// function to house all commmands to do with idx motor 

FUNCTION_BLOCK IDXMotor
VAR_INPUT
	//
END_VAR
VAR_OUTPUT
END_VAR
VAR
	Axis: AXIS_REF;
	Enabled: BOOL := FALSE;
	Override: LREAL:=100;
	MotorError AT%I*	:WORD;
	MotorErrorSent : WORD;
	AxisErrorSent:UDINT;
	NCError : WORD;
	fbMessage : FB_TcMessage;
	EnableEventSent:BOOL:= TRUE;
	HomeEventSent:BOOL:=TRUE;
    fbAxisMoveAbsolute: MC_MoveAbsolute;	
	fbMcHome: MC_Home;
	fbAxisPower: MC_Power;
	fbReset: MC_Reset;
	fbMoveRel : MC_MoveRelative;
	
END_VAR

Axis.ReadStatus();

// cyclic events below 

IF NOT (MotorError = MotorErrorSent) THEN// Creates Event 
	MotorErrorSent:= MotorError;
	fbMessage.CreateEx(TC_Events.LinearMotor.IDXmotorError,0);
	fbMessage.ipArguments.Clear().AddDWord(MotorError);
	fbMessage.Send(0);
END_IF

IF NOT (Axis.NcToPlc.ErrorCode = AxisErrorSent) THEN// Creates Event 
	AxisErrorSent:= Axis.NcToPlc.ErrorCode;
	fbMessage.CreateEx(TC_Events.LinearMotor.AxisError,0);
	fbMessage.ipArguments.Clear().AddDWord(Axis.NcToPlc.ErrorCode);
	fbMessage.Send(0);
END_IF

METHOD PUBLIC Enable : BOOL
VAR_INPUT
EnableMotor :BOOL;
END_VAR
	fbAxisPower( // use in idx class
    Axis:= Axis,
    Enable:= EnableMotor,
    Enable_Positive:= EnableMotor,
    Enable_Negative:= EnableMotor,
    Override:= Override,
	Status=>Enable,
	Error=>
);
	
	
IF EnableMotor = EnableEventSent THEN	
	EnableEventSent := NOT EnableEventSent;
IF EnableMotor THEN
	fbMessage.CreateEx(TC_Events.LinearMotor.Motor_enabled,0);
ELSE
	fbMessage.CreateEx(TC_Events.LinearMotor.Motor_disabled,0);
END_IF
fbMessage.Send(0);
END_IF
END_METHOD

METHOD Estop : BOOL
VAR_INPUT
END_VAR
//stop motor mc stop
END_METHOD

METHOD FB_init : BOOL
VAR_INPUT
	bInitRetains : BOOL; // if TRUE, the retain variables are initialized (warm start / cold start)
	bInCopyCode : BOOL;  // if TRUE, the instance afterwards gets moved into the copy code (online change)
	//AXIS_REF :REFERENCE TO AXIS_REF;
END_VAR
//Axis :=AXIS_REF;
fbMessage.CreateEx(TC_Events.LinearMotor.PLC_restarted,0);
	fbMessage.Send(0);
END_METHOD

METHOD PUBLIC Home : BOOL
VAR_IN_OUT
	Execute:BOOL;
END_VAR
VAR
	HomingDone:BOOL;
	HomingError:BOOL;
	HomingErrorID:UDINT;
END_VAR
// try changing limits to no error mode then home 


	fbMcHome(
	Axis:=Axis,
	Execute:=Execute,
	Position:=510,
	HomingMode:=MC_DefaultHoming,
	Busy=>Home,
	Done=>HomingDone,
	Error=> HomingError,
	ErrorID=> HomingErrorID
);
	
IF Execute THEN
	HomeEventSent:= FALSE;
	fbMessage.CreateEx(TC_Events.LinearMotor.Homing,0);
	fbMessage.Send(0);
	Execute:= FALSE;	
END_IF
IF HomingDone THEN
	fbMessage.CreateEx(TC_Events.LinearMotor.HomingComplete,0);
	fbMessage.Send(0);
END_IF

IF HomingError THEN
	fbMessage.CreateEx(TC_Events.LinearMotor.HomingFailed,0);
	fbMessage.ipArguments.Clear().AddDWord(HomingErrorID);
	fbMessage.Send(0);
END_IF
END_METHOD

METHOD PUBLIC Homed : BOOL
VAR_INPUT
END_VAR
Homed:=Axis.NcToPlc.StateDWord.1;
END_METHOD

METHOD MoveRelative : BOOL
VAR_INPUT
	Distance: LREAL;
	Velocity: LREAL;	
END_VAR
VAR_IN_OUT
	Execute: BOOL;
END_VAR
	fbMoveRel( // in idx class 
    Axis:= Axis,
    Execute:= Execute,
    Distance:= Distance,
    Velocity:= Velocity,);
	
		IF Execute THEN
	fbMessage.CreateEx(TC_Events.LinearMotor.RelativeMove,0);
	fbMessage.ipArguments.Clear();
	fbMessage.ipArguments.AddLReal(Distance);
	fbMessage.ipArguments.AddLReal(Velocity);
	fbMessage.Send(0);
	Execute := FALSE;
END_IF

IF fbMoveRel.Done  THEN
	fbMessage.CreateEx(TC_Events.LinearMotor.MoveComplete,0);
	fbMessage.Send(0);
	
END_IF
END_METHOD

METHOD MoveTo : BOOL
VAR_INPUT
	Position: LREAL;
	Velocity: LREAL;	
END_VAR
VAR_IN_OUT
		Execute: BOOL;
END_VAR
	fbAxisMoveAbsolute( // in idx class 
    Axis:= Axis,
    Execute:= Execute,
    Position:= Position,
    Velocity:= Velocity,);
	
	IF Execute THEN
	fbMessage.CreateEx(TC_Events.LinearMotor.MotorMove,0);
	fbMessage.ipArguments.Clear();
	fbMessage.ipArguments.AddLReal(Position);
	fbMessage.ipArguments.AddLReal(Velocity);
	fbMessage.Send(0);
	Execute := FALSE;

END_IF

IF fbAxisMoveAbsolute.Done  THEN
	fbMessage.CreateEx(TC_Events.LinearMotor.MoveComplete,0);
	fbMessage.Send(0);

	
END_IF
END_METHOD

METHOD Position : LReal
VAR_INPUT
END_VAR
Position:= Axis.NcToPlc.ActPos;
END_METHOD

METHOD Reset : BOOL
VAR_IN_OUT
	ResetAxis:BOOL;
	IDXControlByte1 :USINT;
END_VAR
fbReset(
Axis:=Axis,
Execute:=ResetAxis,
Done =>Reset);

IF resetAxis THEN
IDXControlByte1 := 16#80;// restop linear Motor
fbMessage.CreateEx(TC_Events.LinearMotor.AxisReset,0);
fbMessage.send(0);
resetAxis := FALSE;
END_IF
END_METHOD

METHOD SetSpeed : BOOL
VAR_INPUT
END_VAR
END_METHOD

METHOD PUBLIC Status : ST_AxisStatus
VAR_INPUT
END_VAR
Status := Axis.Status;
END_METHOD

END_FUNCTION_BLOCK

(* stored: Version 1.1.0.1, ProductVersion 3.1.4024.11
   POU IDXMotor: Id {2d0ab0a1-a5a3-4c64-bc51-ecb0c0b67505}, SpecialFunc None
   Method Enable: Id {6ca24d5a-5a8e-43ff-a8c3-908b75374a87}
   Method Estop: Id {ac352b5d-b443-47be-8d49-18781876fd67}
   Method FB_init: Id {98ef687f-1654-43bd-b72b-b96bfe4346b9}
   Method Home: Id {dadfc02e-e1cb-43e2-bcd9-54c8e8b7850a}
   Method Homed: Id {c1cc68f4-37cf-40df-838e-d05e58b07ab5}
   Method MoveRelative: Id {b8493f8e-43b3-46fb-816b-e627b7c74ccc}
   Method MoveTo: Id {08282b44-b328-422b-9de4-f7d3248d3805}
   Method Position: Id {ff434356-d1e2-4881-8909-8666bf1f21d4}
   Method Reset: Id {452ee707-d051-4151-ab20-88e260d22e2a}
   Method SetSpeed: Id {50ebda3b-70f1-42c9-9731-437c5d2aad8f}
   Method Status: Id {f73b2d03-d3bf-443e-8d2d-9005fec7bb7e} *)
